ABB RobotStudio station: UiS_E458_nov18_3_20210919-181048.rsstn

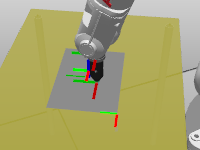
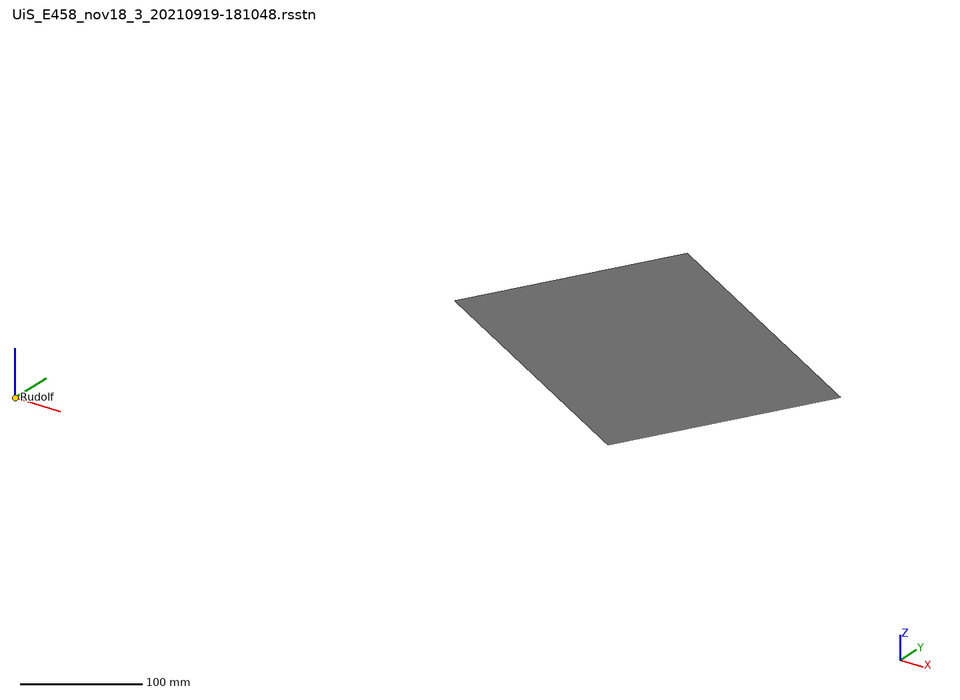
[picture v1: parts stored in the station drawn from their meshes, with robot base, taught points and paths (robot models come from the ABB library and are not in the file)]
Station UiS_E458_nov18_3 (saved by RobotStudio 21.2.9526.0)
Controller Rudolf, task T_ROB1: task frame (RAPID world) sits at (10, 680, 720) mm, rotated rx 0 ry 0 rz -30 deg in the station
Controller Rudolf
  mechanical unit ROB_1: Rudolf, 6 joints, base frame (0, 0, 0) mm
Layout (positions relative to the parent item):
  - PedestalR [part, from Libraries\Pedestal.rslib] at (10, 680, 0) mm, rotated rx 0 ry 0 rz 150 deg
  - Conveyor [part, from Libraries\Conveyor.rslib] at (-998.97, -64.27, 615.81) mm, rotated rx 90 ry 0 rz -90 deg
  - Windowtable [part], size 500 x 2400 x 20 mm
  - TableR [part, from Libraries\Desk.rslib] at (193.4, 1497.66, 0) mm, rotated rx 0 ry 0 rz -120 deg
  - UISpenholder [mechanism, from Libraries\UISpenholder.rslib] at (348.92, 1027.03, 848.1) mm, rotated rx 180 ry 0 rz 150 deg
  - Rudolf [mechanism, from Robots\IRB140_6_81_C_G_03.rslib] at (10, 680, 720) mm, rotated rx 0 ry 0 rz -30 deg; joint values [1.3208, 0.9734, 0.2832, 0, 0.3142, 1.3208] (rad or m)
  - A4Sheet [part] at (209.14, 1020.92, 728.1) mm, rotated rx 0 ry 0 rz -30 deg, size 297 x 210 x 0 mm
Attachment: TableR is attached to PedestalR
Attachment: wobjA4 is attached to A4Sheet
Attachment: UISpenholder is attached to Rudolf / Link6
Station signals: DI doClose, DI doOpen
Station logic (signal -> signal, property => property):
  Norbert.doOpen -> SC_Gripper.diOpen
  Norbert.doClose -> SC_Gripper.diClose
  SC_Gripper.doClosed -> Norbert.diClosed
Targets, tools, work objects and paths stored in the station, written as RAPID:
! task T_ROB1
MODULE E458PenTest
  PERS tooldata tSimplePen:=[TRUE,[[0,0,110],[1,0,0,0]],[1,[0,0,1],[1,0,0,0],0,0,0]];
  TASK PERS wobjdata wobjTableR:=[FALSE,TRUE,"",[[150,500,8],[1,0,0,0]],[[0,0,0],[1,0,0,0]]];
  TASK PERS wobjdata wobjA4:=[FALSE,TRUE,"",[[150,500,8.1],[1,0,0,0]],[[0,0,0],[1,0,0,0]]];
  PERS tooldata UISpenholder:=[TRUE,[[0,0,110],[1,0,0,0]],[1,[0,0,1],[1,0,0,0],0,0,0]];
  CONST robtarget Target_10:=[[0,0,30],[0,0,1,0],[0,0,0,0],[9E+09,9E+09,9E+09,9E+09,9E+09,9E+09]];
  CONST robtarget Target_20:=[[-148.5,-105,0],[0,0,1,0],[0,0,0,0],[9E+09,9E+09,9E+09,9E+09,9E+09,9E+09]];
  PROC main()
  ENDPROC
  PROC Path_10()
  ENDPROC
  PROC section24a()
  ENDPROC
ENDMODULE

! task T_ROB1
MODULE LINKEDM
  PROC Linked_m()
  ENDPROC
ENDMODULE

